# EPICS autosave request: iocs/jungfrauIOC/iocBoot/iocJungfrau/auto_settings.req
file "slsDetector_settings.req",    P=$(P),  R=cam1:
file "NDStdArrays_settings.req",    P=$(P),  R=image1:
#file "commonPlugin_settings.req",   P=$(P)
